PROGRAM HbotForwardKinematics
VAR
	rCurrentY : REAL;
	rCurrentX : REAL;
	
	HMIX : REAL;
	HMIY : REAL;
	
	currentpos : Pos;
	len : ULINT := 4000;
	hist : ARRAY[1..1, 0..4000] OF Pos;
	i : ULINT;
	timer : TON;
	fbAms : FB_GetLocalAmsNetId;
	bReqStarted : BOOL := TRUE;
END_VAR

// calculating real time positions based on axes A and B
rCurrentX := (-GVL.StepperReferenceA.NcToPlc.ActPos - GVL.StepperReferenceB.NcToPlc.ActPos)/2;
rCurrentY := (-GVL.StepperReferenceA.NcToPlc.ActPos + GVL.StepperReferenceB.NcToPlc.ActPos)/2;
HMIX := Round2dp(rCurrentX);
HMIY := Round2dp(rCurrentY);

// keeping historical positions
// ========Step 1, create scruct=======
currentpos.x := rCurrentX;
currentpos.y := rCurrentY;

// ========Step 2, every 0.5 seconds, set new data to be index 0, and do a SHIFT command to the right=======
timer(IN := TRUE, PT := T#0.5S);
IF timer.Q THEN
	hist[1,0] := currentpos;
	FOR i := len-1 TO 1 BY -1 DO
	  hist[1,i] := hist[1,i-1];
	END_FOR 
	timer(IN := FALSE);
END_IF
// ===========================================================================
// =========Just to get local ams net id for python script========
IF bReqStarted THEN
	fbAms(bExecute := TRUE, tTimeOut := T#2S);
	IF NOT fbAms.bBusy THEN
		fbAms(bExecute := FALSE);
		bReqStarted := FALSE;
	END_IF
END_IF

METHOD Round2dp : REAL
VAR_INPUT
	rNum : REAL;
END_VAR
Round2dp := INT_TO_REAL(REAL_TO_INT(rNum * 100))/100;
END_METHOD

END_PROGRAM

(* stored: Version 1.1.0.1, ProductVersion 3.1.4024.11
   POU HbotForwardKinematics: Id {a648ff5d-ed23-4927-a7f3-d9a41701dedb}, SpecialFunc None
   Method Round2dp: Id {a335797a-07b5-47dd-b2fc-d48bdd863733} *)
